// TIA Portal V20 export
// export: Created 2026-07-16T12:59:02.3506962Z, ExportSetting WithDefaults, DisplayName Totally Integrated Automation Portal, DisplayVersion V20 Update 5, DisplayName TIA Portal Openness, DisplayVersion V20 Update 4, DisplayName TIA Portal Version Control Interface, DisplayVersion V20 Update 5, DisplayName SINAMICS Startdrive Advanced, DisplayVersion V20, DisplayName SINAMICS DCC, DisplayVersion V20, DisplayName SINAMICS Startdrive G130, G150, S120, S150, SINAMICS MV, G220, S200, S210, DisplayVersion V20, DisplayName SINAMICS Startdrive G110M, G120, G120C, G120D, G120P, G115D, DisplayVersion V20, DisplayName STEP 7 Professional, DisplayVersion V20 Update 5, DisplayName STEP 7 Safety, DisplayVersion V20 Update 2, DisplayName WinCC Basic/Comfort/Advanced, DisplayVersion V20 Update 5, DisplayName WinCC Unified, DisplayVersion V20 Update 5
FUNCTION_BLOCK "FB_ShredderSequencer"   // FB8, LAD
TITLE = Shredder Plant Sequencer
{ S7_Optimized_Access := 'TRUE' }
VERSION : 0.1
// Shredder plant sequencer (C-118-C-125): commands the shredder motor (via FB_MotorFwdRevSystem, wired at FC_ControlMain) and gates infeed/discharge conveyors and upstream enable, through a stepped cycle. Step legend (C-120): 0=Idle (stopped, waiting for a start condition) - 10=PreStart (siren warning before motion) - 20=DischargeStart (discharge conveyor starting, timed) - 30=ReverseRun (shredder commanded reverse - see FB_MotorFwdRevSystem's own pause/reversal handling) - 40=WaitForwardRun (waiting for forward-run feedback) - 50=Running (normal production; infeed/upstream-enable timers and overcurrent detection are live) - 60=OvercurrentAbort (tripped - pause, then retry into ReverseRun, or stay out if too many reversals).
// stored: AutoNumber true, IsIECCheckEnabled false, IsRetainMemResEnabled false, MemoryReserve 100, SetENOAutomatically false, UDAEnableTagReadback false
   VAR RETAIN
      IO { S7_SetPoint := 'True'} : "UDT_ShredderSequencerIO";   // Caller-visible interface (C-115) - FC_ControlMain writes CycleStart/CycleStop/feedback/tunables in, reads Run*/EnableUpstream/PreStartSounder/motor-command bits out. See the block header for the Step value legend.
   END_VAR
   VAR
      StopCmd : Bool;   // Loss of DownstreamRunning stops the shredder too, not just an operator CycleStop - nowhere for shredded material to go otherwise. Read by every step's own stop transition below.
      ReversalWindowTimeMS : DInt;
      PreStartSounderTimeMS : DInt;
      DischargeConveyorTimeoutMS : DInt;
      ShredderReverseRunTimeMS : DInt;
      InfeedRestartDelayMS : DInt;
      InfeedToUpstreamEnableDelayMS : DInt;
      OvercurrentSpinUpAllowanceMS : DInt;
      OvercurrentMediumDelayMS : DInt;
      OvercurrentHighDelayMS : DInt;
      ReversalRetryPauseTimeMS : DInt;
      ReversalWindowTimer { S7_SetPoint := 'True'} : TON_TIME;
      ReversalStepEdge : Bool;
      ReversalStepEdgeMem : Bool;
      ReversalCount : Int;   // Reversals since the window last re-armed (not per-cycle, unlike the pusher's own PressureTripCount) - ReversalWindowTimer restarts the window every time this is above zero, so ReversalCountThreshold reversals must occur within one ReversalWindowTime of each other to raise ShredderBlockedFault, not just ReversalCountThreshold times ever.
      PreStartTimer { S7_SetPoint := 'True'} : TON_TIME;
      DischargeStartTimer { S7_SetPoint := 'True'} : TON_TIME;
      ReverseRunTimer { S7_SetPoint := 'True'} : TON_TIME;
      InfeedRestartTimer { S7_SetPoint := 'True'} : TON_TIME;
      UpstreamEnableTimer { S7_SetPoint := 'True'} : TON_TIME;
      InfeedRunning : Bool;   // Latched once InfeedRestartTimer has timed out from the last hopper-clear - drives RunInfeedConv directly and (after a further UpstreamEnableTimer delay) EnableUpstream.
      SpinUpTimer { S7_SetPoint := 'True'} : TON_TIME;
      OvercurrentMediumTimer { S7_SetPoint := 'True'} : TON_TIME;
      OvercurrentHighTimer { S7_SetPoint := 'True'} : TON_TIME;
      OvercurrentTripped : Bool;   // KNOWN GAP, not wired to real current yet: both timers below are gated 'AND NOT AlwaysTrue' (permanently false placeholders) because DB_AnalogInput.ShredderMotorCurrent > DB_Settings.OvercurrentSetpointMedium/High is a genuine Real-vs-Real comparison this converter's synthesizer can't type correctly yet (hardcodes Int) - flagged and deferred rather than guessed at. This bit, and Step 50's own overcurrent-abort transition, are dead code until that's built.
      OvercurrentAbortPauseTimer { S7_SetPoint := 'True'} : TON_TIME;
   END_VAR
   VAR_TEMP
      "Time" : Real;
   END_VAR
BEGIN

REGION Network 1: Stop Command
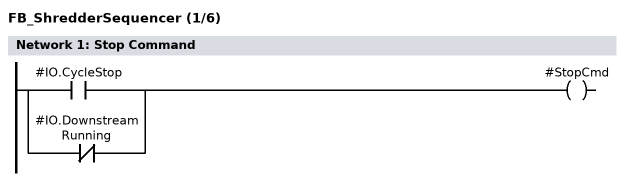
   RUNG wire#powerrail
      Contact( #IO.CycleStop )
      wire#w1
      Coil( #StopCmd )
   END_RUNG
   RUNG wire#powerrail
      I_Contact( #IO.DownstreamRunning )
   END_RUNG wire#w1
   // the same network as SCL:
   #StopCmd := #IO.CycleStop OR NOT #IO.DownstreamRunning;
END_REGION

REGION Network 2: HMI Time Conversions
   // HMI/DB_Settings times are Real seconds for operator legibility; every TON below needs its PT in DInt ms - one MUL+CONVERT pair per timer, matching the MotorDOL FTTime/EnableUPSTime idiom. Kept as one block up front rather than repeated at each timer, so the x1000 idiom is visibly consistent and only ever done once.
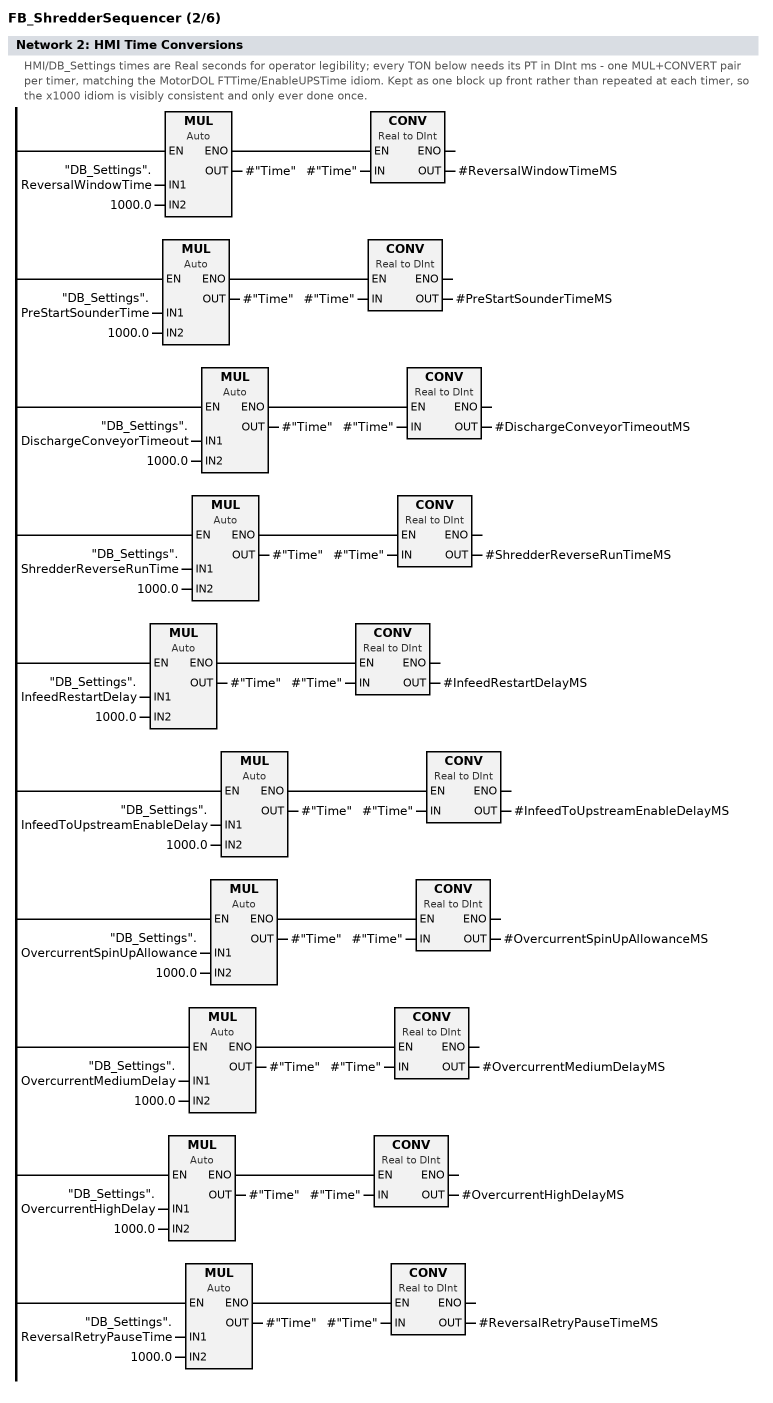
   RUNG wire#powerrail
      Mul(in1 := "DB_Settings".ReversalWindowTime, in2 := 1000.0, out => #"Time")
      { S7_Templates := "[SrcType := Real, DestType := DInt]" } Convert(in := #"Time", out => #ReversalWindowTimeMS)
   END_RUNG
   RUNG wire#powerrail
      Mul(in1 := "DB_Settings".PreStartSounderTime, in2 := 1000.0, out => #"Time")
      { S7_Templates := "[SrcType := Real, DestType := DInt]" } Convert(in := #"Time", out => #PreStartSounderTimeMS)
   END_RUNG
   RUNG wire#powerrail
      Mul(in1 := "DB_Settings".DischargeConveyorTimeout, in2 := 1000.0, out => #"Time")
      { S7_Templates := "[SrcType := Real, DestType := DInt]" } Convert(in := #"Time", out => #DischargeConveyorTimeoutMS)
   END_RUNG
   RUNG wire#powerrail
      Mul(in1 := "DB_Settings".ShredderReverseRunTime, in2 := 1000.0, out => #"Time")
      { S7_Templates := "[SrcType := Real, DestType := DInt]" } Convert(in := #"Time", out => #ShredderReverseRunTimeMS)
   END_RUNG
   RUNG wire#powerrail
      Mul(in1 := "DB_Settings".InfeedRestartDelay, in2 := 1000.0, out => #"Time")
      { S7_Templates := "[SrcType := Real, DestType := DInt]" } Convert(in := #"Time", out => #InfeedRestartDelayMS)
   END_RUNG
   RUNG wire#powerrail
      Mul(in1 := "DB_Settings".InfeedToUpstreamEnableDelay, in2 := 1000.0, out => #"Time")
      { S7_Templates := "[SrcType := Real, DestType := DInt]" } Convert(in := #"Time", out => #InfeedToUpstreamEnableDelayMS)
   END_RUNG
   RUNG wire#powerrail
      Mul(in1 := "DB_Settings".OvercurrentSpinUpAllowance, in2 := 1000.0, out => #"Time")
      { S7_Templates := "[SrcType := Real, DestType := DInt]" } Convert(in := #"Time", out => #OvercurrentSpinUpAllowanceMS)
   END_RUNG
   RUNG wire#powerrail
      Mul(in1 := "DB_Settings".OvercurrentMediumDelay, in2 := 1000.0, out => #"Time")
      { S7_Templates := "[SrcType := Real, DestType := DInt]" } Convert(in := #"Time", out => #OvercurrentMediumDelayMS)
   END_RUNG
   RUNG wire#powerrail
      Mul(in1 := "DB_Settings".OvercurrentHighDelay, in2 := 1000.0, out => #"Time")
      { S7_Templates := "[SrcType := Real, DestType := DInt]" } Convert(in := #"Time", out => #OvercurrentHighDelayMS)
   END_RUNG
   RUNG wire#powerrail
      Mul(in1 := "DB_Settings".ReversalRetryPauseTime, in2 := 1000.0, out => #"Time")
      { S7_Templates := "[SrcType := Real, DestType := DInt]" } Convert(in := #"Time", out => #ReversalRetryPauseTimeMS)
   END_RUNG
   // the same network as SCL:
   #"Time" := "DB_Settings".ReversalWindowTime * 1000.0;
   #ReversalWindowTimeMS := REAL_TO_DINT(#"Time");
   #"Time" := "DB_Settings".PreStartSounderTime * 1000.0;
   #PreStartSounderTimeMS := REAL_TO_DINT(#"Time");
   #"Time" := "DB_Settings".DischargeConveyorTimeout * 1000.0;
   #DischargeConveyorTimeoutMS := REAL_TO_DINT(#"Time");
   #"Time" := "DB_Settings".ShredderReverseRunTime * 1000.0;
   #ShredderReverseRunTimeMS := REAL_TO_DINT(#"Time");
   #"Time" := "DB_Settings".InfeedRestartDelay * 1000.0;
   #InfeedRestartDelayMS := REAL_TO_DINT(#"Time");
   #"Time" := "DB_Settings".InfeedToUpstreamEnableDelay * 1000.0;
   #InfeedToUpstreamEnableDelayMS := REAL_TO_DINT(#"Time");
   #"Time" := "DB_Settings".OvercurrentSpinUpAllowance * 1000.0;
   #OvercurrentSpinUpAllowanceMS := REAL_TO_DINT(#"Time");
   #"Time" := "DB_Settings".OvercurrentMediumDelay * 1000.0;
   #OvercurrentMediumDelayMS := REAL_TO_DINT(#"Time");
   #"Time" := "DB_Settings".OvercurrentHighDelay * 1000.0;
   #OvercurrentHighDelayMS := REAL_TO_DINT(#"Time");
   #"Time" := "DB_Settings".ReversalRetryPauseTime * 1000.0;
   #ReversalRetryPauseTimeMS := REAL_TO_DINT(#"Time");
END_REGION

REGION Network 3: Reversal Re-Arm Window Timer
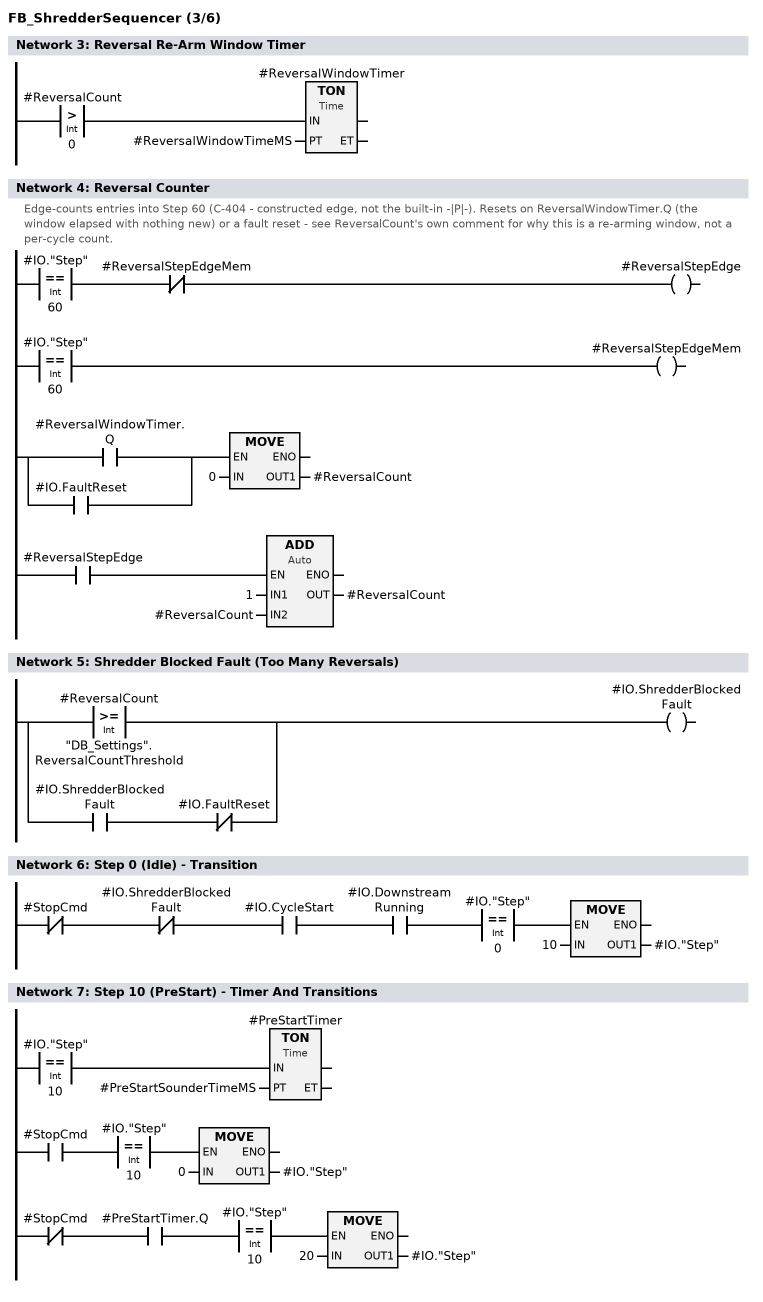
   RUNG wire#powerrail
      { S7_Templates := "SrcType := Int" } GT_Contact(in1 := #ReversalCount, in2 := 0)
      { S7_Templates := "time_type := Time" } #ReversalWindowTimer.TON(pt := #ReversalWindowTimeMS, et =>)
   END_RUNG
   // the same network as SCL:
   #ReversalWindowTimer(IN := #ReversalCount > 0, PT := #ReversalWindowTimeMS);   // TON
END_REGION

REGION Network 4: Reversal Counter
   // Edge-counts entries into Step 60 (C-404 - constructed edge, not the built-in -|P|-). Resets on ReversalWindowTimer.Q (the window elapsed with nothing new) or a fault reset - see ReversalCount's own comment for why this is a re-arming window, not a per-cycle count.
   RUNG wire#powerrail
      { S7_Templates := "SrcType := Int" } EQ_Contact(in1 := #IO."Step", in2 := 60)
      I_Contact( #ReversalStepEdgeMem )
      Coil( #ReversalStepEdge )
   END_RUNG
   RUNG wire#powerrail
      { S7_Templates := "SrcType := Int" } EQ_Contact(in1 := #IO."Step", in2 := 60)
      Coil( #ReversalStepEdgeMem )
   END_RUNG
   RUNG wire#powerrail
      Contact( #ReversalWindowTimer.Q )
      wire#w1
      Move(in := 0, out1 => #ReversalCount)
   END_RUNG
   RUNG wire#powerrail
      Contact( #IO.FaultReset )
   END_RUNG wire#w1
   RUNG wire#powerrail
      Contact( #ReversalStepEdge )
      Add(in1 := 1, in2 := #ReversalCount, out => #ReversalCount)
   END_RUNG
   // the same network as SCL:
   #ReversalStepEdge := (#IO."Step" = 60) AND NOT #ReversalStepEdgeMem;
   #ReversalStepEdgeMem := #IO."Step" = 60;
   IF #ReversalWindowTimer.Q OR #IO.FaultReset THEN #ReversalCount := 0; END_IF;
   IF #ReversalStepEdge THEN #ReversalCount := 1 + #ReversalCount; END_IF;
END_REGION

REGION Network 5: Shredder Blocked Fault (Too Many Reversals)
   RUNG wire#powerrail
      { S7_Templates := "SrcType := Int" } GE_Contact(in1 := #ReversalCount, in2 := "DB_Settings".ReversalCountThreshold)
      wire#w1
      Coil( #IO.ShredderBlockedFault )
   END_RUNG
   RUNG wire#powerrail
      Contact( #IO.ShredderBlockedFault )
      I_Contact( #IO.FaultReset )
   END_RUNG wire#w1
   // the same network as SCL:
   #IO.ShredderBlockedFault := (#ReversalCount >= "DB_Settings".ReversalCountThreshold) OR (#IO.ShredderBlockedFault AND NOT #IO.FaultReset);
END_REGION

REGION Network 6: Step 0 (Idle) - Transition
   RUNG wire#powerrail
      I_Contact( #StopCmd )
      I_Contact( #IO.ShredderBlockedFault )
      Contact( #IO.CycleStart )
      Contact( #IO.DownstreamRunning )
      { S7_Templates := "SrcType := Int" } EQ_Contact(in1 := #IO."Step", in2 := 0)
      Move(in := 10, out1 => #IO."Step")
   END_RUNG
   // the same network as SCL:
   IF NOT #StopCmd AND NOT #IO.ShredderBlockedFault AND #IO.CycleStart AND #IO.DownstreamRunning AND (#IO."Step" = 0) THEN
       #IO."Step" := 10;
   END_IF;
END_REGION

REGION Network 7: Step 10 (PreStart) - Timer And Transitions
   RUNG wire#powerrail
      { S7_Templates := "SrcType := Int" } EQ_Contact(in1 := #IO."Step", in2 := 10)
      { S7_Templates := "time_type := Time" } #PreStartTimer.TON(pt := #PreStartSounderTimeMS, et =>)
   END_RUNG
   RUNG wire#powerrail
      Contact( #StopCmd )
      { S7_Templates := "SrcType := Int" } EQ_Contact(in1 := #IO."Step", in2 := 10)
      Move(in := 0, out1 => #IO."Step")
   END_RUNG
   RUNG wire#powerrail
      I_Contact( #StopCmd )
      Contact( #PreStartTimer.Q )
      { S7_Templates := "SrcType := Int" } EQ_Contact(in1 := #IO."Step", in2 := 10)
      Move(in := 20, out1 => #IO."Step")
   END_RUNG
   // the same network as SCL:
   #PreStartTimer(IN := #IO."Step" = 10, PT := #PreStartSounderTimeMS);   // TON
   IF #StopCmd AND (#IO."Step" = 10) THEN #IO."Step" := 0; END_IF;
   IF NOT #StopCmd AND #PreStartTimer.Q AND (#IO."Step" = 10) THEN #IO."Step" := 20; END_IF;
END_REGION

REGION Network 8: Step 20 (DischargeStart) - Timer, Timeout Fault, And Transitions
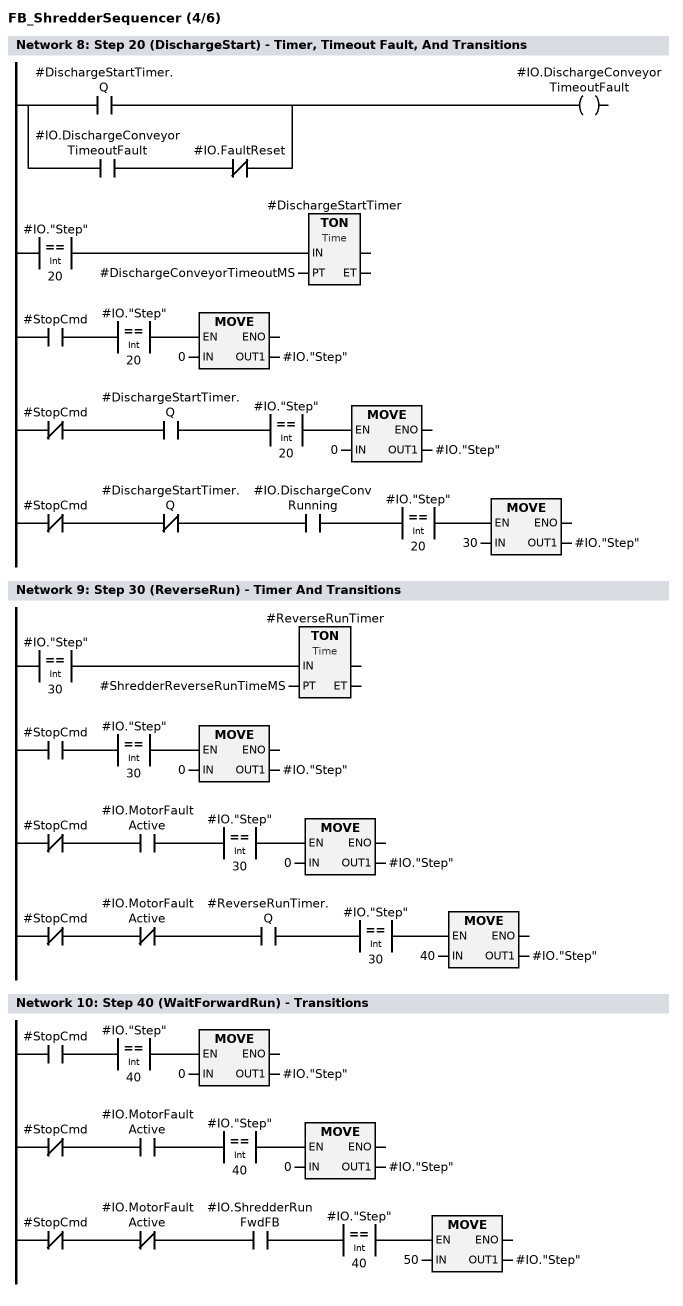
   RUNG wire#powerrail
      Contact( #DischargeStartTimer.Q )
      wire#w1
      Coil( #IO.DischargeConveyorTimeoutFault )
   END_RUNG
   RUNG wire#powerrail
      Contact( #IO.DischargeConveyorTimeoutFault )
      I_Contact( #IO.FaultReset )
   END_RUNG wire#w1
   RUNG wire#powerrail
      { S7_Templates := "SrcType := Int" } EQ_Contact(in1 := #IO."Step", in2 := 20)
      { S7_Templates := "time_type := Time" } #DischargeStartTimer.TON(pt := #DischargeConveyorTimeoutMS, et =>)
   END_RUNG
   RUNG wire#powerrail
      Contact( #StopCmd )
      { S7_Templates := "SrcType := Int" } EQ_Contact(in1 := #IO."Step", in2 := 20)
      Move(in := 0, out1 => #IO."Step")
   END_RUNG
   RUNG wire#powerrail
      I_Contact( #StopCmd )
      Contact( #DischargeStartTimer.Q )
      { S7_Templates := "SrcType := Int" } EQ_Contact(in1 := #IO."Step", in2 := 20)
      Move(in := 0, out1 => #IO."Step")
   END_RUNG
   RUNG wire#powerrail
      I_Contact( #StopCmd )
      I_Contact( #DischargeStartTimer.Q )
      Contact( #IO.DischargeConvRunning )
      { S7_Templates := "SrcType := Int" } EQ_Contact(in1 := #IO."Step", in2 := 20)
      Move(in := 30, out1 => #IO."Step")
   END_RUNG
   // the same network as SCL:
   #IO.DischargeConveyorTimeoutFault := #DischargeStartTimer.Q OR (#IO.DischargeConveyorTimeoutFault AND NOT #IO.FaultReset);
   #DischargeStartTimer(IN := #IO."Step" = 20, PT := #DischargeConveyorTimeoutMS);   // TON
   IF #StopCmd AND (#IO."Step" = 20) THEN #IO."Step" := 0; END_IF;
   IF NOT #StopCmd AND #DischargeStartTimer.Q AND (#IO."Step" = 20) THEN #IO."Step" := 0; END_IF;
   IF NOT #StopCmd AND NOT #DischargeStartTimer.Q AND #IO.DischargeConvRunning AND (#IO."Step" = 20) THEN
       #IO."Step" := 30;
   END_IF;
END_REGION

REGION Network 9: Step 30 (ReverseRun) - Timer And Transitions
   RUNG wire#powerrail
      { S7_Templates := "SrcType := Int" } EQ_Contact(in1 := #IO."Step", in2 := 30)
      { S7_Templates := "time_type := Time" } #ReverseRunTimer.TON(pt := #ShredderReverseRunTimeMS, et =>)
   END_RUNG
   RUNG wire#powerrail
      Contact( #StopCmd )
      { S7_Templates := "SrcType := Int" } EQ_Contact(in1 := #IO."Step", in2 := 30)
      Move(in := 0, out1 => #IO."Step")
   END_RUNG
   RUNG wire#powerrail
      I_Contact( #StopCmd )
      Contact( #IO.MotorFaultActive )
      { S7_Templates := "SrcType := Int" } EQ_Contact(in1 := #IO."Step", in2 := 30)
      Move(in := 0, out1 => #IO."Step")
   END_RUNG
   RUNG wire#powerrail
      I_Contact( #StopCmd )
      I_Contact( #IO.MotorFaultActive )
      Contact( #ReverseRunTimer.Q )
      { S7_Templates := "SrcType := Int" } EQ_Contact(in1 := #IO."Step", in2 := 30)
      Move(in := 40, out1 => #IO."Step")
   END_RUNG
   // the same network as SCL:
   #ReverseRunTimer(IN := #IO."Step" = 30, PT := #ShredderReverseRunTimeMS);   // TON
   IF #StopCmd AND (#IO."Step" = 30) THEN #IO."Step" := 0; END_IF;
   IF NOT #StopCmd AND #IO.MotorFaultActive AND (#IO."Step" = 30) THEN #IO."Step" := 0; END_IF;
   IF NOT #StopCmd AND NOT #IO.MotorFaultActive AND #ReverseRunTimer.Q AND (#IO."Step" = 30) THEN
       #IO."Step" := 40;
   END_IF;
END_REGION

REGION Network 10: Step 40 (WaitForwardRun) - Transitions
   RUNG wire#powerrail
      Contact( #StopCmd )
      { S7_Templates := "SrcType := Int" } EQ_Contact(in1 := #IO."Step", in2 := 40)
      Move(in := 0, out1 => #IO."Step")
   END_RUNG
   RUNG wire#powerrail
      I_Contact( #StopCmd )
      Contact( #IO.MotorFaultActive )
      { S7_Templates := "SrcType := Int" } EQ_Contact(in1 := #IO."Step", in2 := 40)
      Move(in := 0, out1 => #IO."Step")
   END_RUNG
   RUNG wire#powerrail
      I_Contact( #StopCmd )
      I_Contact( #IO.MotorFaultActive )
      Contact( #IO.ShredderRunFwdFB )
      { S7_Templates := "SrcType := Int" } EQ_Contact(in1 := #IO."Step", in2 := 40)
      Move(in := 50, out1 => #IO."Step")
   END_RUNG
   // the same network as SCL:
   IF #StopCmd AND (#IO."Step" = 40) THEN #IO."Step" := 0; END_IF;
   IF NOT #StopCmd AND #IO.MotorFaultActive AND (#IO."Step" = 40) THEN #IO."Step" := 0; END_IF;
   IF NOT #StopCmd AND NOT #IO.MotorFaultActive AND #IO.ShredderRunFwdFB AND (#IO."Step" = 40) THEN
       #IO."Step" := 50;
   END_IF;
END_REGION

REGION Network 11: Step 50 (Running) - Infeed Restart, Upstream Enable, And Outputs
   // UpstreamEnableTimer's own IN reads InfeedRunning one scan behind this network's own InfeedRunning update below (it's kind-ordered before the coil that writes it) - harmless for a multi-second delay, and matches this design's original timing exactly. EnableUpstream lives here, next to its own timer, rather than in the general Output Commands network - this is the output the MotorFwdRevSystem CALL-site correction was specifically about: it must only ever come from Step=50 dwell time, never from motor-running telemetry.
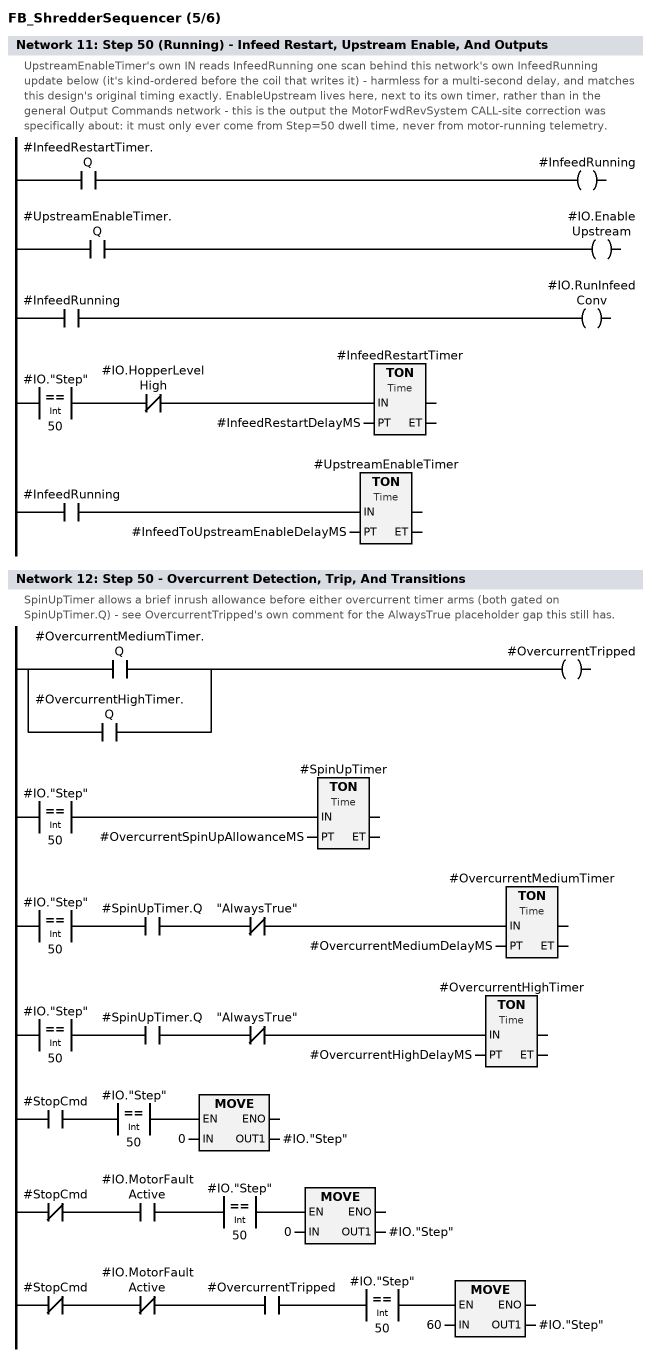
   RUNG wire#powerrail
      Contact( #InfeedRestartTimer.Q )
      Coil( #InfeedRunning )
   END_RUNG
   RUNG wire#powerrail
      Contact( #UpstreamEnableTimer.Q )
      Coil( #IO.EnableUpstream )
   END_RUNG
   RUNG wire#powerrail
      Contact( #InfeedRunning )
      Coil( #IO.RunInfeedConv )
   END_RUNG
   RUNG wire#powerrail
      { S7_Templates := "SrcType := Int" } EQ_Contact(in1 := #IO."Step", in2 := 50)
      I_Contact( #IO.HopperLevelHigh )
      { S7_Templates := "time_type := Time" } #InfeedRestartTimer.TON(pt := #InfeedRestartDelayMS, et =>)
   END_RUNG
   RUNG wire#powerrail
      Contact( #InfeedRunning )
      { S7_Templates := "time_type := Time" } #UpstreamEnableTimer.TON(pt := #InfeedToUpstreamEnableDelayMS, et =>)
   END_RUNG
   // the same network as SCL:
   #InfeedRunning := #InfeedRestartTimer.Q;
   #IO.EnableUpstream := #UpstreamEnableTimer.Q;
   #IO.RunInfeedConv := #InfeedRunning;
   #InfeedRestartTimer(IN := (#IO."Step" = 50) AND NOT #IO.HopperLevelHigh, PT := #InfeedRestartDelayMS);   // TON
   #UpstreamEnableTimer(IN := #InfeedRunning, PT := #InfeedToUpstreamEnableDelayMS);   // TON
END_REGION

REGION Network 12: Step 50 - Overcurrent Detection, Trip, And Transitions
   // SpinUpTimer allows a brief inrush allowance before either overcurrent timer arms (both gated on SpinUpTimer.Q) - see OvercurrentTripped's own comment for the AlwaysTrue placeholder gap this still has.
   RUNG wire#powerrail
      Contact( #OvercurrentMediumTimer.Q )
      wire#w1
      Coil( #OvercurrentTripped )
   END_RUNG
   RUNG wire#powerrail
      Contact( #OvercurrentHighTimer.Q )
   END_RUNG wire#w1
   RUNG wire#powerrail
      { S7_Templates := "SrcType := Int" } EQ_Contact(in1 := #IO."Step", in2 := 50)
      { S7_Templates := "time_type := Time" } #SpinUpTimer.TON(pt := #OvercurrentSpinUpAllowanceMS, et =>)
   END_RUNG
   RUNG wire#powerrail
      { S7_Templates := "SrcType := Int" } EQ_Contact(in1 := #IO."Step", in2 := 50)
      Contact( #SpinUpTimer.Q )
      I_Contact( "AlwaysTrue" )
      { S7_Templates := "time_type := Time" } #OvercurrentMediumTimer.TON(pt := #OvercurrentMediumDelayMS, et =>)
   END_RUNG
   RUNG wire#powerrail
      { S7_Templates := "SrcType := Int" } EQ_Contact(in1 := #IO."Step", in2 := 50)
      Contact( #SpinUpTimer.Q )
      I_Contact( "AlwaysTrue" )
      { S7_Templates := "time_type := Time" } #OvercurrentHighTimer.TON(pt := #OvercurrentHighDelayMS, et =>)
   END_RUNG
   RUNG wire#powerrail
      Contact( #StopCmd )
      { S7_Templates := "SrcType := Int" } EQ_Contact(in1 := #IO."Step", in2 := 50)
      Move(in := 0, out1 => #IO."Step")
   END_RUNG
   RUNG wire#powerrail
      I_Contact( #StopCmd )
      Contact( #IO.MotorFaultActive )
      { S7_Templates := "SrcType := Int" } EQ_Contact(in1 := #IO."Step", in2 := 50)
      Move(in := 0, out1 => #IO."Step")
   END_RUNG
   RUNG wire#powerrail
      I_Contact( #StopCmd )
      I_Contact( #IO.MotorFaultActive )
      Contact( #OvercurrentTripped )
      { S7_Templates := "SrcType := Int" } EQ_Contact(in1 := #IO."Step", in2 := 50)
      Move(in := 60, out1 => #IO."Step")
   END_RUNG
   // the same network as SCL:
   #OvercurrentTripped := #OvercurrentMediumTimer.Q OR #OvercurrentHighTimer.Q;
   #SpinUpTimer(IN := #IO."Step" = 50, PT := #OvercurrentSpinUpAllowanceMS);   // TON
   #OvercurrentMediumTimer(IN := (#IO."Step" = 50) AND #SpinUpTimer.Q AND NOT "AlwaysTrue",   // TON
                           PT := #OvercurrentMediumDelayMS);
   #OvercurrentHighTimer(IN := (#IO."Step" = 50) AND #SpinUpTimer.Q AND NOT "AlwaysTrue",   // TON
                         PT := #OvercurrentHighDelayMS);
   IF #StopCmd AND (#IO."Step" = 50) THEN #IO."Step" := 0; END_IF;
   IF NOT #StopCmd AND #IO.MotorFaultActive AND (#IO."Step" = 50) THEN #IO."Step" := 0; END_IF;
   IF NOT #StopCmd AND NOT #IO.MotorFaultActive AND #OvercurrentTripped AND (#IO."Step" = 50) THEN
       #IO."Step" := 60;
   END_IF;
END_REGION

REGION Network 13: Step 60 (OvercurrentAbort) - Timer And Transitions
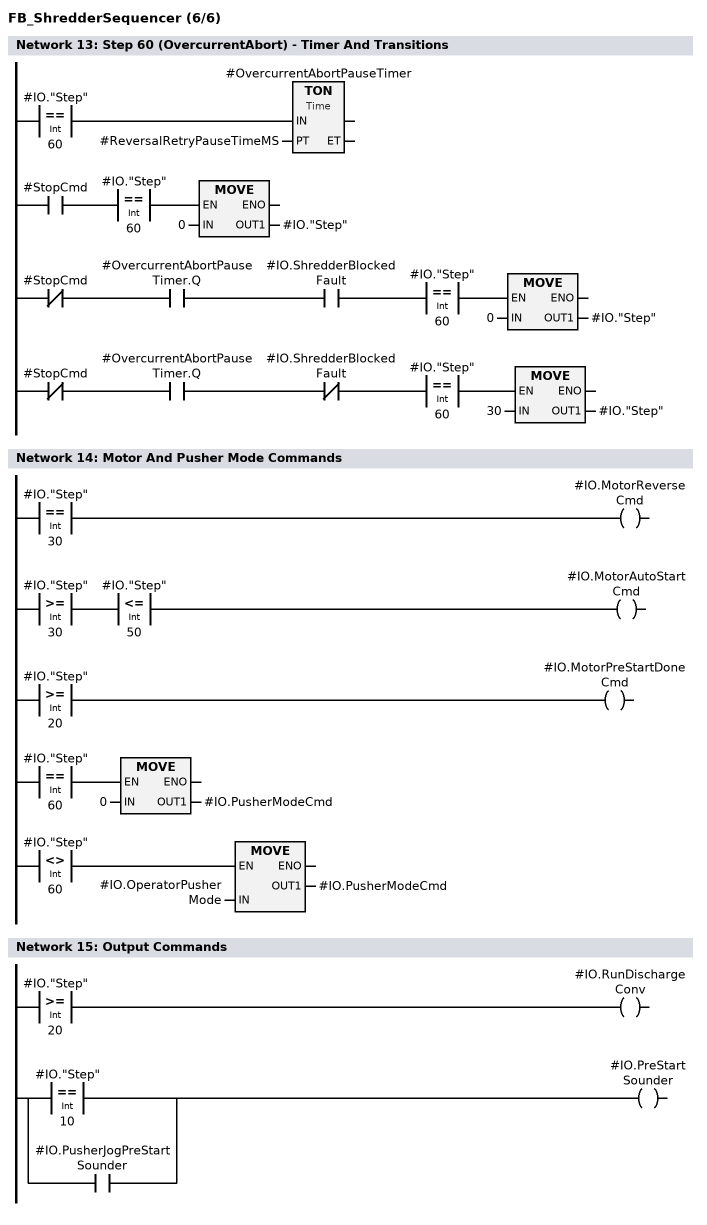
   RUNG wire#powerrail
      { S7_Templates := "SrcType := Int" } EQ_Contact(in1 := #IO."Step", in2 := 60)
      { S7_Templates := "time_type := Time" } #OvercurrentAbortPauseTimer.TON(pt := #ReversalRetryPauseTimeMS, et =>)
   END_RUNG
   RUNG wire#powerrail
      Contact( #StopCmd )
      { S7_Templates := "SrcType := Int" } EQ_Contact(in1 := #IO."Step", in2 := 60)
      Move(in := 0, out1 => #IO."Step")
   END_RUNG
   RUNG wire#powerrail
      I_Contact( #StopCmd )
      Contact( #OvercurrentAbortPauseTimer.Q )
      Contact( #IO.ShredderBlockedFault )
      { S7_Templates := "SrcType := Int" } EQ_Contact(in1 := #IO."Step", in2 := 60)
      Move(in := 0, out1 => #IO."Step")
   END_RUNG
   RUNG wire#powerrail
      I_Contact( #StopCmd )
      Contact( #OvercurrentAbortPauseTimer.Q )
      I_Contact( #IO.ShredderBlockedFault )
      { S7_Templates := "SrcType := Int" } EQ_Contact(in1 := #IO."Step", in2 := 60)
      Move(in := 30, out1 => #IO."Step")
   END_RUNG
   // the same network as SCL:
   #OvercurrentAbortPauseTimer(IN := #IO."Step" = 60, PT := #ReversalRetryPauseTimeMS);   // TON
   IF #StopCmd AND (#IO."Step" = 60) THEN #IO."Step" := 0; END_IF;
   IF NOT #StopCmd AND #OvercurrentAbortPauseTimer.Q AND #IO.ShredderBlockedFault AND (#IO."Step" = 60) THEN
       #IO."Step" := 0;
   END_IF;
   IF NOT #StopCmd AND #OvercurrentAbortPauseTimer.Q AND NOT #IO.ShredderBlockedFault AND (#IO."Step" = 60) THEN
       #IO."Step" := 30;
   END_IF;
END_REGION

REGION Network 14: Motor And Pusher Mode Commands
   RUNG wire#powerrail
      { S7_Templates := "SrcType := Int" } EQ_Contact(in1 := #IO."Step", in2 := 30)
      Coil( #IO.MotorReverseCmd )
   END_RUNG
   RUNG wire#powerrail
      { S7_Templates := "SrcType := Int" } GE_Contact(in1 := #IO."Step", in2 := 30)
      { S7_Templates := "SrcType := Int" } LE_Contact(in1 := #IO."Step", in2 := 50)
      Coil( #IO.MotorAutoStartCmd )
   END_RUNG
   RUNG wire#powerrail
      { S7_Templates := "SrcType := Int" } GE_Contact(in1 := #IO."Step", in2 := 20)
      Coil( #IO.MotorPreStartDoneCmd )
   END_RUNG
   RUNG wire#powerrail
      { S7_Templates := "SrcType := Int" } EQ_Contact(in1 := #IO."Step", in2 := 60)
      Move(in := 0, out1 => #IO.PusherModeCmd)
   END_RUNG
   RUNG wire#powerrail
      { S7_Templates := "SrcType := Int" } NE_Contact(in1 := #IO."Step", in2 := 60)
      Move(in := #IO.OperatorPusherMode, out1 => #IO.PusherModeCmd)
   END_RUNG
   // the same network as SCL:
   #IO.MotorReverseCmd := #IO."Step" = 30;
   #IO.MotorAutoStartCmd := (#IO."Step" >= 30) AND (#IO."Step" <= 50);
   #IO.MotorPreStartDoneCmd := #IO."Step" >= 20;
   IF #IO."Step" = 60 THEN #IO.PusherModeCmd := 0; END_IF;
   IF #IO."Step" <> 60 THEN #IO.PusherModeCmd := #IO.OperatorPusherMode; END_IF;
END_REGION

REGION Network 15: Output Commands
   RUNG wire#powerrail
      { S7_Templates := "SrcType := Int" } GE_Contact(in1 := #IO."Step", in2 := 20)
      Coil( #IO.RunDischargeConv )
   END_RUNG
   RUNG wire#powerrail
      { S7_Templates := "SrcType := Int" } EQ_Contact(in1 := #IO."Step", in2 := 10)
      wire#w1
      Coil( #IO.PreStartSounder )
   END_RUNG
   RUNG wire#powerrail
      Contact( #IO.PusherJogPreStartSounder )
   END_RUNG wire#w1
   // the same network as SCL:
   #IO.RunDischargeConv := #IO."Step" >= 20;
   #IO.PreStartSounder := (#IO."Step" = 10) OR #IO.PusherJogPreStartSounder;
END_REGION
END_FUNCTION_BLOCK
